// TIA Portal V19 export
FUNCTION_BLOCK "FP_Saeure.GP0x"   // FB1001, LAD
TITLE = Filterpumpe Säure
{ S7_Optimized_Access := 'TRUE' }
// Funktionen:  Filternn / /Filterwechsel / Spülen
// stored: AutoNumber false, MemoryReserve 100, SetENOAutomatically false
   VAR RETAIN
      In { ExternalAccessible := 'False'; ExternalVisible := 'False'; ExternalWritable := 'False'} : Struct
         NotHalt : Bool;
         ext_Freigabe : Bool;   // Kein Gasalarm, Kein Notstrom
         Auto : Bool;   // Paneltaste
         Ein : Bool;   // Paneltaste
         Quitt_FW : Bool;   // Paneltaste
         FU_betriebsbereit : Bool;
         FU_Stoerung : Bool;
         Niv_TLS : Bool;
         Niv_min : Bool;
         Niv_max : Bool;
         Niv_Uel : Bool;
         Frg_Niv_CM05 : Bool;
         Leckage_ok : Bool;
         SRM_Saugseite_auf : Bool;
         SRM_Saugseite_zu : Bool;
         SRM_Eingang_Filter_auf : Bool;
         SRM_Eingang_Filter_zu : Bool;
         SRM_Ausgang_Filter_auf : Bool;
         SRM_Ausgang_Filter_zu : Bool;
         SRM_Entluften_auf : Bool;
         SRM_Entlueften_zu : Bool;
         SRM_Eingang_Spülltg_P_auf : Bool;   // Pumpe
         SRM_Eingang_Spülltg_P_zu : Bool;   // Pumpe
         SRM_Eingang_Spülltg_F_auf : Bool;   // Filter
         SRM_Eingang_Spülltg_F_zu : Bool;   // Filter
         SRM_Ausgang_Spülltg_auf : Bool;
         SRM_Ausgang_Spülltg_zu : Bool;
         Sensor_FG_links : Bool;
         Sensor_FG_rechts : Bool;
         Einhausung_HQ0x_zu : Bool;
         GW_p_FP : Bool;
         GW_p_FG : Bool;
         GW_LF_FP : Bool;
         Betriebsart : USInt := 0;   // Paneltaste
         FU_speed : Int;
         Druck_Pumpe : Real;
         Delta_p_Filter : Real;
      END_STRUCT;
      Param { ExternalAccessible := 'False'; ExternalVisible := 'False'; ExternalWritable := 'False'} : Struct
         SW_Hand : Int;   // [%]
         SW_Auto_AZ : Int;   // [%]
         SW_Auto_aAZ : Int;   // [%]
         Spülzeit_Pumpe : Time;
         FG_Zeit_leeren_Saurebecken : Time;
         FG_Zeit_leeren_CM05 : Time;
         FW_Spülzeit : Time;
         FW_Wartezeit : Time;
         FW_Zeit_fuellen : Time;
         DT_Druckaufbau : Time;
         DT_Testzeit_Pumpe : Time;
         DT_Testzeit_Filter : Time;
         SW_Drucktest_Pumpe : Real;
         SW_Drucktest_Filter : Real;
         WarnGr_FW : Real;
         Wechsel_FW : Real;
         Name_Pumpe : String[12];
         Name_Filter : String[12];
      END_STRUCT;
      Zst { ExternalAccessible := 'False'; ExternalVisible := 'False'; ExternalWritable := 'False'} : Struct
         Status_GP0x : USInt;
         Status_FW : USInt;
         Status_DT_Pumpe : USInt;
         Status_DT_Filter : USInt;
         Restzeit_Spülen_Pumpe : Time;
         Restzeit_Filter : Time;
         Restzeit_DT : Time;
         Spuelen_Pumpe : Bool;
         Spuelen_Filter : Bool;
         Spuelen_aktiv : Bool;
         Drucktest_aktiv : Bool;
         Filtern : Bool;
         Zeit_laeuft : Bool;
         Drucktest_Pu_ok : Bool;
         Drucktest_Filter_ok : Bool;
         Bedienung_erlaubt : Bool;
         speed : Int;   // [%]
      END_STRUCT;
      Mld { ExternalAccessible := 'False'; ExternalVisible := 'False'; ExternalWritable := 'False'} : Struct
         Leckage : Bool;
         GW_p_FP : Bool;
         GW_LF_FP : Bool;
         GW_p_FG : Bool;
         FG_links_nicht_zu : Bool;
         FG_rechts_nicht_zu : Bool;
         Einhausung_nicht_zu : Bool;
         FU_nicht_bereit : Bool;
         FU_Stoerung : Bool;
         FG_Spülen_Ende : Bool;
         n_Auto : Bool;
         TO_Druckaufbau : Bool;
         Drucktest_Pumpe_ok : Bool;
         Drucktest_Pumpe_Fehler : Bool;
         Pu_Spuelen_Fertig : Bool;
         Drucktest_Filter_ok : Bool;
         Drucktest_Filter_Fehler : Bool;
         Drucktest_Filter_erfordert : Bool;
         Filterbeutel_Wechsel_Vorwarngrenze : Bool;
         Filterbeutel_Wechsel_notwendig : Bool;
      END_STRUCT;
      Out { ExternalAccessible := 'False'; ExternalVisible := 'False'; ExternalWritable := 'False'} : Struct
         GP0x_Ein : Bool;
         Ventil_Saugseite : Bool;
         Ventil_Eingang_Filter : Bool;
         Ventil_Ausgang_Filter : Bool;
         Ventil_Entlueften : Bool;
         Spülventil_P_Eingang : Bool;
         Spülventil_F_Eingang : Bool;
         Spülventil_Ausgang : Bool;
         Soll_speed : Int;
      END_STRUCT;
   END_VAR
   VAR
      IEC_Timer { ExternalAccessible := 'False'; ExternalVisible := 'False'; ExternalWritable := 'False'} : Struct
         Spülen_Pumpe { S7_SetPoint := 'True'} : TP_TIME;
         Filterwechsel { S7_SetPoint := 'True'} : TP_TIME;
         GW_p { S7_SetPoint := 'True'} : TON_TIME;
         Drucktest { S7_SetPoint := 'True'} : TP_TIME;
         TO_Druckaufbau { S7_SetPoint := 'True'} : TON_TIME;
         Verz_Ueberdruck { S7_SetPoint := 'True'} : TON_TIME;
         Spülventil_Ausgang { S7_SetPoint := 'True'} : TOF_TIME;
      END_STRUCT;
      R_TRIG_Hand_EIN { ExternalAccessible := 'False'; ExternalVisible := 'False'; ExternalWritable := 'False'} : R_TRIG;
   END_VAR
   VAR_TEMP
      Spülzeit_Pumpe : Time;
      Spülzeit_Filter : Time;
      Zeit_DT : Time;
      posFl_Hand : Bool;
      Filtergehäuse_ok : Bool;
   END_VAR
   VAR CONSTANT
      Niv_TLS : USInt := 2;
      Niv_Min : USInt := 20;
      Niv_max : USInt := 90;
      Niv_Uel : USInt := 98;
      S0 : USInt := 0;
      S1 : USInt := 1;
      S2 : USInt := 2;
      S3 : USInt := 3;
      S4 : USInt := 4;
      S5 : USInt := 5;
      S6 : USInt := 6;
      S7 : USInt := 7;
      S8 : USInt := 8;
      S10_FG_Leeren : USInt := 10;
   END_VAR
BEGIN

REGION Network 1 (SCL): Input
   // Panelbedienung und Sensoren --> Input()

    // positive Flanke "Hand Ein"
   #R_TRIG_Hand_EIN(CLK := #In.Ein,
                    Q => #posFl_Hand);
END_REGION

REGION Network 2 (SCL): Ansteuerung
   // Filtergehäuse geschlossen
   #Filtergehäuse_ok := #In.Sensor_FG_links AND #In.Sensor_FG_rechts AND #In.Einhausung_HQ0x_zu;

   // Alles AUS
   IF (#In.Betriebsart = 2) AND #In.Leckage_ok AND #In.ext_Freigabe THEN // Spülen
       // Ausschaltverzögert - Druckabbau
       #IEC_Timer.Spülventil_Ausgang(IN := #Out.Spülventil_P_Eingang,
                                     PT := T#3s,
                                     Q => #Out.Spülventil_Ausgang);
   ELSE
       #Out.Spülventil_P_Eingang := FALSE;
       #Out.Spülventil_Ausgang := FALSE;
   END_IF;
   #Out.Spülventil_F_Eingang := FALSE;
   #Zst.Restzeit_Spülen_Pumpe := T#0s;
   #Zst.Restzeit_Filter := T#0s;
   #Out.Ventil_Saugseite := FALSE;
   #Out.Ventil_Eingang_Filter := FALSE;
   #Out.Ventil_Entlueften := FALSE;
   #Out.Ventil_Ausgang_Filter := FALSE;

   // "Normal"-Betrieb
   #Zst.Bedienung_erlaubt := NOT #In.Ein AND NOT #In.Auto AND NOT #Mld.Drucktest_Pumpe_Fehler AND NOT #Mld.Drucktest_Filter_Fehler;

   //Drucktest Pumpe rücksetzen
   IF #In.Betriebsart <> 3 OR #Zst.Spuelen_aktiv OR #Zst.Filtern OR NOT #In.Ein THEN
       #Mld.Drucktest_Pumpe_ok := FALSE;
       // #Mld.Drucktest_Pumpe_Fehler := FALSE;
       #Zst.Status_DT_Pumpe := 0;
       #Zst.Drucktest_aktiv := FALSE;
   END_IF;
   //Drucktest Filter rücksetzen
   IF #In.Betriebsart <> 4 OR #Zst.Spuelen_aktiv OR #Zst.Filtern OR NOT #In.Ein THEN
       #Mld.Drucktest_Filter_ok := FALSE;
       // #Mld.Drucktest_Filter_Fehler := FALSE;
       #Zst.Status_DT_Filter := 0;
   END_IF;
   IF #In.Betriebsart <> 3 AND #In.Betriebsart <> 4 THEN
       #Mld.TO_Druckaufbau := FALSE;
   END_IF;
   //Filterwechsel rücksetzen
   IF #In.Betriebsart <> 1 OR #Zst.Spuelen_aktiv OR NOT #In.Ein THEN
       #Zst.Status_FW := 0;
   END_IF;
   //Spülmeldung rücksetzen
   IF #In.Betriebsart <> 2 OR NOT #In.Ein THEN
       #Mld.Pu_Spuelen_Fertig := FALSE;
   END_IF;
   IF #In.Leckage_ok AND #In.ext_Freigabe THEN
       CASE #In.Betriebsart OF
           0:  // Filterbetrieb
                         // Ventile öffnen
               IF NOT #Mld.Drucktest_Filter_erfordert AND NOT #Mld.Filterbeutel_Wechsel_notwendig THEN
                   #Out.Ventil_Saugseite := (#In.Auto OR #In.Ein) AND #In.Niv_TLS AND #In.SRM_Ausgang_Spülltg_zu AND #In.SRM_Eingang_Spülltg_P_zu AND #In.SRM_Eingang_Spülltg_F_zu;
                   #Out.Ventil_Eingang_Filter := #Out.Ventil_Saugseite;
                   #Out.Ventil_Ausgang_Filter := #Out.Ventil_Eingang_Filter;
               END_IF;
                   // Wenn geöffnet --> Frg Pumpe
                   #Zst.Filtern := #In.SRM_Eingang_Filter_auf AND #In.SRM_Ausgang_Filter_auf AND #In.SRM_Saugseite_auf;
                   // #Zst.Status_FW := #Ende;

           1:  // Filterwechsel 
               REGION Filterwechsel
                   #Zst.Filtern := FALSE;
                   CASE #Zst.Status_FW OF
                       #S0:  // Grundzustand
                           IF #In.Auto OR #In.Ein THEN
                               #Zst.Status_FW := #S1;
                           END_IF;

                       #S1:    // 1. Mal Leerlaufen ins Säurebecken - vor Spülen: Pumpe Aus - Ventile Auf - Zeit warten
                           // Ventile öffnen
                           #Out.Ventil_Eingang_Filter := #Filtergehäuse_ok AND #In.SRM_Ausgang_Spülltg_zu AND #In.SRM_Eingang_Spülltg_P_zu AND #In.SRM_Eingang_Spülltg_F_zu;
                           #Out.Ventil_Ausgang_Filter := #Out.Ventil_Eingang_Filter;
                           #Out.Ventil_Saugseite := #Out.Ventil_Eingang_Filter;
                           #Out.Ventil_Entlueften := #Out.Ventil_Eingang_Filter;

                           #IEC_Timer.Filterwechsel(IN := #In.SRM_Eingang_Filter_auf AND #In.SRM_Ausgang_Filter_auf AND #In.SRM_Saugseite_auf AND #In.SRM_Entluften_auf,
                                                    PT := #Param.FG_Zeit_leeren_Saurebecken,
                                                    ET => #Spülzeit_Filter,
                                                    Q => #Zst.Zeit_laeuft);
                           #Zst.Restzeit_Filter := #Param.FG_Zeit_leeren_Saurebecken - #Spülzeit_Filter;

                           IF NOT #Zst.Zeit_laeuft AND #In.SRM_Eingang_Filter_auf AND #In.SRM_Ausgang_Filter_auf AND #In.SRM_Saugseite_auf AND #In.SRM_Entluften_auf THEN
                               #Out.Ventil_Ausgang_Filter := #Out.Ventil_Eingang_Filter := #Out.Ventil_Saugseite := #Out.Ventil_Entlueften := FALSE;
                               #Zst.Status_FW := #S2;
                           END_IF;

                       #S2:    // Spülen Filtergehäuse
                           // Ventile öffnen
                           #Out.Spülventil_F_Eingang := #In.Frg_Niv_CM05;
                           #Out.Spülventil_Ausgang := NOT #Out.Ventil_Entlueften;
                           #Out.Ventil_Entlueften := #Zst.Zeit_laeuft AND #Zst.Restzeit_Filter < T#15s; //#Spülzeit_Filter > T#45s AND #Spülzeit_Filter <= T#60s;
                           #IEC_Timer.Filterwechsel(IN := #In.SRM_Ausgang_Spülltg_auf AND #In.SRM_Eingang_Spülltg_F_auf,
                                                    PT := #Param.FW_Spülzeit,
                                                    ET => #Spülzeit_Filter,
                                                    Q => #Zst.Zeit_laeuft);
                           #Zst.Restzeit_Filter := #Param.FW_Spülzeit - #Spülzeit_Filter;

                           IF NOT #Zst.Zeit_laeuft AND #In.SRM_Ausgang_Spülltg_auf AND #In.SRM_Eingang_Spülltg_F_auf THEN
                               #Out.Spülventil_F_Eingang := #Out.Spülventil_Ausgang := FALSE;
                               #Out.Ventil_Entlueften := FALSE;
                               #Zst.Status_FW := #S3;
                           END_IF;

                       #S3:    // Warten --> Meldung
                           #IEC_Timer.Filterwechsel(IN := #In.SRM_Ausgang_Spülltg_zu AND #In.SRM_Eingang_Spülltg_F_zu AND #In.SRM_Entlueften_zu,
                                                    PT := #Param.FW_Wartezeit,
                                                    ET => #Spülzeit_Filter,
                                                    Q => #Zst.Zeit_laeuft);
                           #Zst.Restzeit_Filter := #Param.FW_Wartezeit - #Spülzeit_Filter;
                           // Ventile öffnen
                           IF #Zst.Zeit_laeuft AND #Zst.Restzeit_Filter < t#10s THEN
                               #Out.Ventil_Entlueften := TRUE;// #Zst.Zeit_laeuft AND #Zst.Restzeit_Filter < t#10s; // #Spülzeit_Filter > T#45s AND #Spülzeit_Filter <= T#60s;
                               #Out.Spülventil_F_Eingang := #Out.Ventil_Entlueften;
                           ELSE
                               #Out.Ventil_Entlueften := FALSE;
                               #Out.Spülventil_F_Eingang := FALSE;
                           END_IF;

                           IF NOT #Zst.Zeit_laeuft AND #In.SRM_Eingang_Spülltg_F_auf AND #In.SRM_Entluften_auf THEN
                               #Zst.Status_FW := #S4;
                           END_IF;

                       #S4:    // 2. Mal Leerlaufen in CM05 - nach Spülen: Pumpe Aus - Ventile Auf - Zeit warten
                           // Ventile öffnen
                           #Out.Ventil_Saugseite := FALSE;
                         //  #Out.Ventil_Eingang_Filter := FALSE;  04.08.21
                           #Out.Spülventil_Ausgang :=  #In.Frg_Niv_CM05 (*AND #In.SRM_Ausgang_Filter_zu 04.08.21*) AND #In.SRM_Eingang_Spülltg_P_zu AND #In.SRM_Eingang_Spülltg_F_zu;
                           #Out.Ventil_Entlueften := #Out.Spülventil_Ausgang;

                           #IEC_Timer.Filterwechsel(IN :=  #In.Frg_Niv_CM05 (*AND #In.SRM_Eingang_Filter_zu 04.08.21*) AND #In.SRM_Ausgang_Spülltg_auf AND #In.SRM_Saugseite_zu AND #In.SRM_Entluften_auf,
                                                    PT := #Param.FG_Zeit_leeren_CM05,
                                                    ET => #Spülzeit_Filter,
                                                    Q => #Zst.Zeit_laeuft);
                           #Zst.Restzeit_Filter := #Param.FG_Zeit_leeren_CM05 - #Spülzeit_Filter;

                           // 03.08.21
                           //Eine Bitte habe ich noch, zwar beim Filterwechsel. Es steht immer noch recht viel restliches saures Wasser im Behälter,
                           //könntest du bitte für den letzten Schritt noch 10sec für HQ01 den QM23 und bei HQ02 den QM60 öffnen.
                           //Somit ist auch die Leitung zur Leitfähigkeitsmessung leer.
                           #Out.Ventil_Eingang_Filter := #Out.Ventil_Ausgang_Filter := #Zst.Zeit_laeuft AND #Zst.Restzeit_Filter <= t#40s;// 03.08.21

                           IF NOT #Zst.Zeit_laeuft (*AND #In.SRM_Eingang_Filter_zu 04.08.21*) AND #In.SRM_Ausgang_Spülltg_auf AND #In.SRM_Saugseite_zu AND #In.SRM_Entluften_auf THEN
                               #Out.Ventil_Ausgang_Filter := #Out.Ventil_Eingang_Filter := #Out.Ventil_Saugseite := #Out.Ventil_Entlueften := FALSE;
                               #Zst.Status_FW := #S5;
                               #Mld.FG_Spülen_Ende := TRUE;
                           END_IF;

                       #S5:    // man.Wechsel --> Quittierung
                           // Ventile bleiben offen --> Nachlauf Restwasser in CM05
                           #Out.Ventil_Saugseite := FALSE;
                           #Out.Ventil_Eingang_Filter := FALSE;
                           #Out.Spülventil_Ausgang := #In.Frg_Niv_CM05 AND #In.SRM_Ausgang_Filter_zu AND #In.SRM_Eingang_Spülltg_P_zu AND #In.SRM_Eingang_Spülltg_F_zu;
                           #Out.Ventil_Entlueften := #Out.Spülventil_Ausgang;

                           IF #Filtergehäuse_ok AND #In.Quitt_FW THEN
                               #Mld.FG_Spülen_Ende := FALSE;
                               #Mld.Drucktest_Filter_erfordert := TRUE;
                               #Mld.Filterbeutel_Wechsel_notwendig := FALSE;
                               #In.Quitt_FW := FALSE;
                               #Zst.Status_FW := #S8;
                           END_IF;

                           (*     
                            #S6:    //Filtergehäuse füllen
                                #Out.Ventil_Saugseite := (#In.Auto OR #In.Ein) AND #In.Niv_TLS AND #In.SRM_Ausgang_Spülltg_zu AND #In.SRM_Eingang_Spülltg_P_zu AND #In.SRM_Eingang_Spülltg_F_zu;
                                #Out.Ventil_Eingang_Filter := #Out.Ventil_Saugseite;
                                #Out.Ventil_Ausgang_Filter := TRUE;
                                #Out.Spülventil_Ausgang := FALSE;

                                // Wenn geöffnet --> Frg Pumpe
                                #IEC_Timer.Filterwechsel(IN := #In.SRM_Eingang_Filter_auf AND #In.SRM_Saugseite_auf AND #In.SRM_Ausgang_Filter_auf,
                                                         PT := #Param.FW_Zeit_fuellen,
                                                         ET => #Spülzeit_Filter,
                                                         Q => #Zst.Zeit_laeuft);

                                #Zst.Filtern := #In.SRM_Eingang_Filter_auf AND #In.SRM_Ausgang_Filter_auf AND #In.SRM_Saugseite_auf;

                                #Zst.Restzeit_Filter := #Param.FW_Zeit_fuellen - #Spülzeit_Filter;

                                IF NOT #Zst.Zeit_laeuft AND #Zst.Filtern THEN
                                    #Zst.Status_FW := #S7;
                                END_IF;


                            #S7:    // Kreislauf öffnen
                                // #Out.Ventil_Ausgang_Filter := TRUE;
                                // #Out.Spülventil_Ausgang := NOT #In.SRM_Ausgang_Filter_auf;

                                // IF #In.SRM_Ausgang_Filter_auf AND #In.SRM_Ausgang_Spülltg_zu THEN
                                //     #Zst.Status_FW := #S8;
                                // END_IF;
                                #Zst.Filtern := FALSE;
                                IF #Zst.speed <= 20 THEN
                                    #Out.Ventil_Saugseite := FALSE;
                                    #Out.Ventil_Eingang_Filter := FALSE;
                                    #Out.Ventil_Ausgang_Filter := FALSE;
                                    #Out.Spülventil_Ausgang := FALSE;
                                END_IF;

                                IF NOT  #Zst.Filtern AND  #In.SRM_Saugseite_zu AND #In.SRM_Eingang_Filter_zu AND #In.SRM_Ausgang_Filter_zu AND #In.SRM_Ausgang_Spülltg_zu THEN
                                    #Zst.Status_FW := #S8;
                                END_IF;
                                  *)
                       #S8: // Ende
                           ;
                   END_CASE;
               END_REGION

           2:// Spülen - nur Hand
               #Zst.Filtern := FALSE;
               #Zst.Status_FW := #S0;

               IF NOT #Mld.Drucktest_Filter_erfordert AND NOT #Mld.Filterbeutel_Wechsel_notwendig THEN
                   IF #In.Ein AND #In.Frg_Niv_CM05 THEN
                       IF #posFl_Hand THEN
                           #Zst.Spuelen_aktiv := TRUE;
                       END_IF;
                       #Out.Spülventil_P_Eingang := #Filtergehäuse_ok AND #In.SRM_Ausgang_Filter_zu AND #In.SRM_Saugseite_zu AND #Zst.Spuelen_aktiv;
                       #Out.Ventil_Eingang_Filter := #Out.Spülventil_Ausgang;

                       #IEC_Timer.Spülen_Pumpe(IN := #In.SRM_Eingang_Spülltg_P_auf AND #In.SRM_Ausgang_Spülltg_auf,
                                               PT := #Param.Spülzeit_Pumpe,
                                               Q => #Zst.Spuelen_Pumpe,
                                               ET => #Spülzeit_Pumpe);
                       #Zst.Restzeit_Spülen_Pumpe := #Param.Spülzeit_Pumpe - #Spülzeit_Pumpe;

                       IF #In.SRM_Eingang_Spülltg_P_auf AND #In.SRM_Ausgang_Spülltg_auf AND NOT #Zst.Spuelen_Pumpe THEN
                           #Zst.Spuelen_aktiv := FALSE;
                           #Out.Spülventil_P_Eingang := FALSE;
                       END_IF;

                       // Fertig
                       IF NOT #Zst.Spuelen_Pumpe AND NOT #Zst.Spuelen_aktiv AND NOT #Out.Spülventil_Ausgang THEN
                           #Out.Spülventil_P_Eingang := FALSE;
                           #Out.Spülventil_Ausgang := FALSE;
                           #Out.Ventil_Eingang_Filter := FALSE;
                           #Zst.Restzeit_Spülen_Pumpe := T#0s;
                           #Mld.Pu_Spuelen_Fertig := TRUE;
                       END_IF;
                   ELSE
                       #Zst.Spuelen_Pumpe := FALSE;
                       #Out.Spülventil_P_Eingang := FALSE;
                       #Out.Spülventil_Ausgang := FALSE;
                       #Out.Ventil_Eingang_Filter := FALSE;
                       #Zst.Restzeit_Spülen_Pumpe := T#0s;
                   END_IF;
                   // Ausschaltverzögert - Druckabbau
                   #IEC_Timer.Spülventil_Ausgang(IN := #Out.Spülventil_P_Eingang,
                                                 PT := T#3s,
                                                 Q => #Out.Spülventil_Ausgang);
               END_IF;
           3: // Spülen + Drucktest - nur Hand
               #Zst.Filtern := FALSE;
               #Zst.Status_FW := #S0;
               IF NOT #Mld.Drucktest_Filter_erfordert AND NOT #Mld.Filterbeutel_Wechsel_notwendig THEN
                   IF NOT #Zst.Drucktest_aktiv THEN
                       IF #In.Ein AND #In.Frg_Niv_CM05 THEN
                           IF #posFl_Hand THEN
                               #Zst.Spuelen_aktiv := TRUE;
                           END_IF;
                           #Out.Spülventil_P_Eingang := #Filtergehäuse_ok AND #In.SRM_Ausgang_Filter_zu AND #In.SRM_Saugseite_zu;
                           #Out.Spülventil_Ausgang := #Out.Spülventil_P_Eingang;
                           #Out.Ventil_Eingang_Filter := #Out.Spülventil_P_Eingang;

                           #IEC_Timer.Spülen_Pumpe(IN := #In.SRM_Eingang_Spülltg_P_auf AND #In.SRM_Ausgang_Spülltg_auf,
                                                   PT := #Param.Spülzeit_Pumpe,
                                                   Q => #Zst.Spuelen_Pumpe,
                                                   ET => #Spülzeit_Pumpe);
                           #Zst.Restzeit_Spülen_Pumpe := #Param.Spülzeit_Pumpe - #Spülzeit_Pumpe;

                           IF #In.SRM_Eingang_Spülltg_P_auf AND #In.SRM_Ausgang_Spülltg_auf AND NOT #Zst.Spuelen_Pumpe THEN
                               #Zst.Spuelen_aktiv := FALSE;
                           END_IF;

                           // Fertig
                           IF NOT #Zst.Spuelen_Pumpe AND NOT #Zst.Spuelen_aktiv THEN
                               #Out.Spülventil_Ausgang := FALSE;
                               #Out.Ventil_Eingang_Filter := FALSE;
                               #Zst.Restzeit_Spülen_Pumpe := T#0s;
                               #Zst.Drucktest_aktiv := TRUE;
                               #Zst.Status_DT_Pumpe := #S1;
                           END_IF;
                       ELSE
                           #Zst.Spuelen_Pumpe := FALSE;
                           #Out.Spülventil_P_Eingang := FALSE;
                           #Out.Spülventil_Ausgang := FALSE;
                           #Out.Ventil_Eingang_Filter := FALSE;
                           #Zst.Restzeit_Spülen_Pumpe := T#0s;
                       END_IF;
                   END_IF;


                   //Drucktest
                   IF #Zst.Drucktest_aktiv THEN

                       CASE #Zst.Status_DT_Pumpe OF
                           #S1:  //Druckaufbau

                               IF "DB_Temporaer".Drucksensoren_deaktiviert THEN //20.01.22
                                   #Zst.Drucktest_Pu_ok := TRUE;

                                   "Ergebnis_DT"("Name" := #Param.Name_Pumpe,
                                                 akt_Zeit := "Uhrzeit".aktDatum,
                                                 ok := #Zst.Drucktest_Pu_ok,
                                                 Fehler := NOT #Zst.Drucktest_Pu_ok);

                                   #Mld.Drucktest_Pumpe_ok := #Zst.Drucktest_Pu_ok;
                                   #Mld.Drucktest_Pumpe_Fehler := NOT #Zst.Drucktest_Pu_ok;

                                   #Zst.Status_DT_Pumpe := #S4;
                               ELSE
                                   #Out.Spülventil_P_Eingang := #In.SRM_Ausgang_Filter_zu AND #In.SRM_Saugseite_zu;
                                   #Out.Ventil_Eingang_Filter := FALSE;
                                   #Out.Spülventil_Ausgang := FALSE;

                                   IF (#In.Druck_Pumpe > #Param.SW_Drucktest_Pumpe + 0.25 AND #In.SRM_Eingang_Filter_zu) OR #Mld.TO_Druckaufbau THEN
                                       #Out.Spülventil_P_Eingang := FALSE;
                                       #Zst.Status_DT_Pumpe := #S2;
                                   END_IF;

                               END_IF;

                           #S2: //Wartezeit
                               #IEC_Timer.Drucktest(IN := #In.SRM_Eingang_Spülltg_P_zu,
                                                    PT := #Param.DT_Testzeit_Pumpe,
                                                    Q => #Zst.Zeit_laeuft,
                                                    ET => #Zeit_DT);
                               #Zst.Restzeit_DT := #Param.DT_Testzeit_Pumpe - #Zeit_DT;

                               IF NOT #Zst.Zeit_laeuft AND #In.SRM_Eingang_Spülltg_P_zu THEN
                                   #Zst.Restzeit_DT := T#0s;
                                   #Zst.Status_DT_Pumpe := #S3;
                               END_IF;

                           #S3:// Überprüfung
                               #Zst.Drucktest_Pu_ok := #In.Druck_Pumpe >= #Param.SW_Drucktest_Pumpe;

                               "Ergebnis_DT"("Name" := #Param.Name_Pumpe,
                                             akt_Zeit := "Uhrzeit".aktDatum,
                                             ok := #Zst.Drucktest_Pu_ok,
                                             Fehler := NOT #Zst.Drucktest_Pu_ok);

                               #Mld.Drucktest_Pumpe_ok := #Zst.Drucktest_Pu_ok;
                               #Mld.Drucktest_Pumpe_Fehler := NOT #Zst.Drucktest_Pu_ok;

                               #Zst.Status_DT_Pumpe := #S4;

                           #S4: // ENDE
                               ;
                       END_CASE;
                   END_IF;
               END_IF;
           4: // Drucktest Filter
               #Zst.Filtern := FALSE;
               IF #posFl_Hand (*AND NOT #Mld.Filterbeutel_Wechsel_notwendig - 23.08.22, falls während Drucktest die Meldung aktiv wird, dass es nicht im deadlock ist*) THEN
                   #Zst.Status_DT_Filter:= 1;
               END_IF;

               CASE #Zst.Status_DT_Filter OF
                   #S1:  //Druckaufbau

                       IF "DB_Temporaer".Drucksensoren_deaktiviert THEN //20.01.22
                           #Zst.Drucktest_Filter_ok := TRUE;

                           "Ergebnis_DT"("Name" := #Param.Name_Filter,
                                         akt_Zeit := "Uhrzeit".aktDatum,
                                         ok := #Zst.Drucktest_Filter_ok,
                                         Fehler := NOT #Zst.Drucktest_Filter_ok);

                           #Mld.Drucktest_Filter_ok := #Zst.Drucktest_Filter_ok;
                           #Mld.Drucktest_Filter_Fehler := NOT #Zst.Drucktest_Filter_ok;
                           #Mld.Drucktest_Filter_erfordert := FALSE;
                           #Zst.Status_DT_Filter := #S10_FG_Leeren;

                       ELSE
                           #Out.Spülventil_F_Eingang := #Filtergehäuse_ok AND #In.SRM_Ausgang_Filter_zu AND #In.SRM_Saugseite_zu;
                           #Out.Ventil_Eingang_Filter := FALSE;
                           #Out.Spülventil_Ausgang := FALSE;

                           IF (ABS(#In.Delta_p_Filter) > #Param.SW_Drucktest_Filter + 0.25 AND #In.SRM_Eingang_Spülltg_F_auf) OR #Mld.TO_Druckaufbau OR #Mld.GW_p_FG THEN
                               #Out.Spülventil_F_Eingang := FALSE;
                               #Zst.Status_DT_Filter := #S2;
                           END_IF;
                           #Zst.Restzeit_DT := #Param.DT_Druckaufbau - #IEC_Timer.TO_Druckaufbau.ET;

                       END_IF;

                   #S2: //Wartezeit
                       #IEC_Timer.Drucktest(IN := #In.SRM_Eingang_Spülltg_F_zu,
                                            PT := #Param.DT_Testzeit_Filter,
                                            Q => #Zst.Zeit_laeuft,
                                            ET => #Zeit_DT);
                       #Zst.Restzeit_DT := #Param.DT_Testzeit_Filter - #Zeit_DT;

                       IF NOT #Zst.Zeit_laeuft AND #In.SRM_Eingang_Spülltg_F_zu THEN
                           #Zst.Restzeit_DT := T#0s;
                           #Zst.Status_DT_Filter := #S3;
                       END_IF;

                   #S3:// Überprüfung
                       #Zst.Drucktest_Filter_ok := ABS(#In.Delta_p_Filter) >= #Param.SW_Drucktest_Filter;

                       "Ergebnis_DT"("Name" := #Param.Name_Filter,
                                     akt_Zeit := "Uhrzeit".aktDatum,
                                     ok := #Zst.Drucktest_Filter_ok,
                                     Fehler := NOT #Zst.Drucktest_Filter_ok);

                       #Mld.Drucktest_Filter_ok := #Zst.Drucktest_Filter_ok;
                       #Mld.Drucktest_Filter_Fehler := NOT #Zst.Drucktest_Filter_ok;
                       #Mld.Drucktest_Filter_erfordert := FALSE;
                       #Zst.Status_DT_Filter := #S10_FG_Leeren;

                   #S10_FG_Leeren: // Filtergehäuse nach NIO Drucktest leeren in CM05
                       // Ventile öffnen
                       #Out.Ventil_Saugseite := FALSE;
                     //#Out.Ventil_Eingang_Filter := FALSE;  04.08.21
                       #Out.Spülventil_Ausgang := #In.Frg_Niv_CM05 (*AND #In.SRM_Ausgang_Filter_zu 04.08.21*) AND #In.SRM_Eingang_Spülltg_P_zu AND #In.SRM_Eingang_Spülltg_F_zu;;
                       #Out.Ventil_Entlueften :=  #Out.Spülventil_Ausgang;

                       #IEC_Timer.Filterwechsel(IN := #In.Frg_Niv_CM05 (*AND #In.SRM_Eingang_Filter_zu04.08.21*)AND #In.SRM_Ausgang_Spülltg_auf AND #In.SRM_Saugseite_zu AND #In.SRM_Entluften_auf,
                                                PT := #Param.FG_Zeit_leeren_CM05,
                                                ET => #Spülzeit_Filter,
                                                Q => #Zst.Zeit_laeuft);
                       #Zst.Restzeit_DT := #Param.FG_Zeit_leeren_CM05 - #Spülzeit_Filter;

                       // 04.08.21
                       //Eine Bitte habe ich noch, zwar beim Filterwechsel. Es steht immer noch recht viel restliches saures Wasser im Behälter,
                       //könntest du bitte für den letzten Schritt noch 10sec für HQ01 den QM23 und bei HQ02 den QM60 öffnen.
                       //Somit ist auch die Leitung zur Leitfähigkeitsmessung leer.
                       #Out.Ventil_Eingang_Filter := #Out.Ventil_Ausgang_Filter := #Zst.Zeit_laeuft AND #Zst.Restzeit_DT <= t#40s;// 03.08.21

                       IF NOT #Zst.Zeit_laeuft (*AND #In.SRM_Eingang_Filter_zu04.08.21*)AND #In.SRM_Ausgang_Spülltg_auf AND #In.SRM_Saugseite_zu AND #In.SRM_Entluften_auf THEN
                           #Out.Spülventil_Ausgang := #Out.Ventil_Eingang_Filter := #Out.Ventil_Saugseite := #Out.Ventil_Entlueften := FALSE;
                           #Zst.Status_DT_Filter := #S4;
                       END_IF;

                   #S4: // ENDE
                       ;


               END_CASE;

       END_CASE;
   END_IF;

       // Pumpe an    
   #Out.GP0x_Ein := #Zst.Filtern AND NOT #In.NotHalt AND #Filtergehäuse_ok AND #In.Leckage_ok AND #In.ext_Freigabe AND (#In.Ein OR #In.Auto);

       // Geschwindigkeitsvorgabe
       // SEW: 100% == 3000 U/min == 15000 Digits
       IF #Out.GP0x_Ein THEN
           IF #In.Ein THEN
               #Out.Soll_speed := #Param.SW_Hand * 150;
           ELSE
               IF "Uhrzeit".AZ_aktiv THEN
                   #Out.Soll_speed := #Param.SW_Auto_AZ * 150;
               ELSE
                   #Out.Soll_speed := #Param.SW_Auto_aAZ * 150;
               END_IF;
           END_IF;
       ELSE
           #Out.Soll_speed := 0;
       END_IF;
END_REGION

REGION Network 3 (SCL): Überwachung / Meldungen
   // Leckage
   #Mld.Leckage := NOT #In.Leckage_ok;

   // Zeitüberschreitung Druckaufbau
   #IEC_Timer.TO_Druckaufbau(IN := #Zst.Status_DT_Pumpe = #S1 OR #Zst.Status_DT_Filter = #S1,
                             PT := #Param.DT_Druckaufbau,
                             Q => #Mld.TO_Druckaufbau);

   //Grenzwert Druck Filtergehäuse
   #IEC_Timer.Verz_Ueberdruck(IN := #In.GW_p_FG,
                              PT :=t#3s,
                              Q => #Mld.GW_p_FG);

   // Nicht geschlossen
   #Mld.Einhausung_nicht_zu := NOT #In.Einhausung_HQ0x_zu;
   #Mld.FG_links_nicht_zu := NOT #In.Sensor_FG_links;
   #Mld.FG_rechts_nicht_zu := NOT #In.Sensor_FG_rechts;

   // Grenzwert Druck Pumpe
   #IEC_Timer.GW_p(IN :=#Out.GP0x_Ein AND #In.GW_p_FP,
                   PT := T#3s,
                   Q => #Mld.GW_p_FP);
   // Grenzwert Leitfähigkeit
   #Mld.GW_LF_FP := #In.GW_LF_FP;

   // Frequenzumrichter 24V-Betrieb
   #Mld.FU_nicht_bereit := NOT #In.FU_betriebsbereit AND NOT #In.NotHalt;
   // Störung Frequenzumrichter
   #Mld.FU_Stoerung := #In.FU_Stoerung AND NOT #In.NotHalt;
   // nicht in Automatik
   #Mld.n_Auto := NOT #In.Auto AND "DB_ANLAGE".BA.Automat_ein;
   // Filterwechsel
   #Mld.Filterbeutel_Wechsel_Vorwarngrenze := #In.Delta_p_Filter > #Param.WarnGr_FW AND NOT #Mld.Filterbeutel_Wechsel_notwendig;

   IF #In.Delta_p_Filter > #Param.Wechsel_FW THEN
       #Mld.Filterbeutel_Wechsel_notwendig := TRUE;
   END_IF;
END_REGION

REGION Network 4 (SCL): --> Visu
   // Status Pumpe
   "Status_E0A"(Hand := #In.Ein,
                Auto := #In.Auto,
                SonderModus_PumpeSpuelen:=#Zst.Spuelen_Pumpe,
                Stoerung := #In.FU_Stoerung OR NOT #In.FU_betriebsbereit,
                Ausgang := #Out.GP0x_Ein,
                StatusByte => #Zst.Status_GP0x);

   // Ist-Geschwindigkeit FU
   // SEW: 100% == 3000 U/min == 15000 Digits
   #Zst.speed := #In.FU_speed / 150; // in[%]
END_REGION
END_FUNCTION_BLOCK
